// TIA Portal project "Project4" (V17)

(* hardware
DEVICE "S7-1200 station_1"  S7-1200 Station
   slot 0: "Rack_0"  S7-1200 Rack  Rack  V1.0
   slot 1: "PLC_1"  CPU 1214C AC/DC/Rly  6ES7 214-1BG40-0XB0  V4.2
*)

// ===== PLC "PLC_1"  CPU 1214C AC/DC/Rly =====

VAR_GLOBAL   // PLC tag table "Default tag table"
   "PB0" AT %I0.0 : Bool;
   "PB1" AT %I0.1 : Bool;
   "PB2" AT %I0.2 : Bool;
   "PB3" AT %I0.3 : Bool;
   "PB4" AT %I0.4 : Bool;
   "PB5" AT %I0.5 : Bool;
   "PL1" AT %Q0.0 : Bool;
   "PL2" AT %Q0.1 : Bool;
   "PL3" AT %Q0.2 : Bool;
   "PL4" AT %Q0.3 : Bool;
   "X1" AT %M0.0 : Bool;
   "X2" AT %M0.1 : Bool;
   "X3" AT %M0.2 : Bool;
   "X4" AT %M0.3 : Bool;
   "X5" AT %M0.4 : Bool;
   "Tag_1" AT %M10.0 : Bool;
END_VAR

ORGANIZATION_BLOCK "Main"   // OB1, LAD, ProgramCycle
TITLE = "Main Program Sweep (Cycle)"
{ S7_Optimized_Access := 'TRUE' }
VERSION : 0.1
   VAR_INPUT
      Initial_Call : Bool;   // Initial call of this OB
      Remanence : Bool;   // =True, if remanent data are available
   END_VAR
   VAR_TEMP   // added for the SCL form of the ladder/FBD networks
      _w1 : Bool;
   END_VAR
BEGIN

REGION Network 1
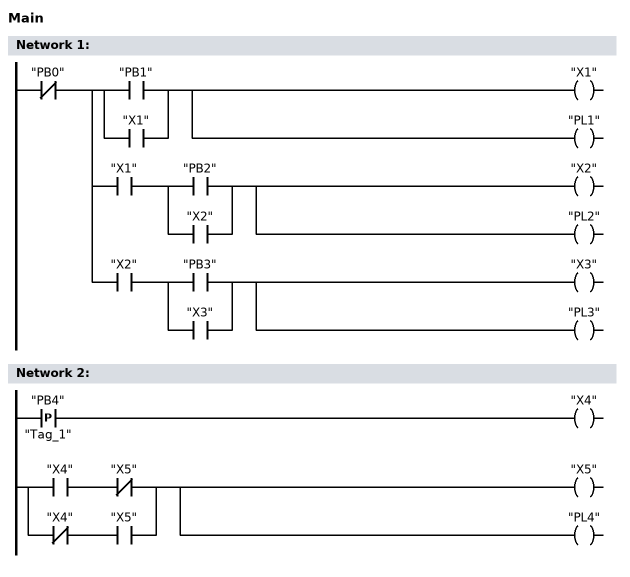
   RUNG wire#powerrail
      I_Contact( "PB0" )
      wire#w1
      Contact( "PB1" )
      wire#w2
      Coil( "X1" )
   END_RUNG
   RUNG wire#w1
      Contact( "X1" )
   END_RUNG wire#w2
   RUNG wire#w2
      Coil( "PL1" )
   END_RUNG
   RUNG wire#w1
      Contact( "X1" )
      wire#w3
      Contact( "PB2" )
      wire#w4
      Coil( "X2" )
   END_RUNG
   RUNG wire#w3
      Contact( "X2" )
   END_RUNG wire#w4
   RUNG wire#w4
      Coil( "PL2" )
   END_RUNG
   RUNG wire#w1
      Contact( "X2" )
      wire#w5
      Contact( "PB3" )
      wire#w6
      Coil( "X3" )
   END_RUNG
   RUNG wire#w5
      Contact( "X3" )
   END_RUNG wire#w6
   RUNG wire#w6
      Coil( "PL3" )
   END_RUNG
   // the same network as SCL:
   "X1" := NOT "PB0" AND ("PB1" OR "X1");
   "PL1" := "X1";
   "X2" := NOT "PB0" AND "X1" AND ("PB2" OR "X2");
   "PL2" := "X2";
   "X3" := NOT "PB0" AND "X2" AND ("PB3" OR "X3");
   "PL3" := "X3";
END_REGION

REGION Network 2
   RUNG wire#powerrail
      P_Contact(operand := "PB4", bit := "Tag_1")
      Coil( "X4" )
   END_RUNG
   RUNG wire#powerrail
      Contact( "X4" )
      I_Contact( "X5" )
      wire#w1
      Coil( "X5" )
   END_RUNG
   RUNG wire#powerrail
      I_Contact( "X4" )
      Contact( "X5" )
   END_RUNG wire#w1
   RUNG wire#w1
      Coil( "PL4" )
   END_RUNG
   // the same network as SCL:
   #_w1 := "PB4" AND NOT "Tag_1";   // rising edge of "PB4"
   "Tag_1" := "PB4";
   "X4" := #_w1;
   "X5" := ("X4" AND NOT "X5") OR (NOT "X4" AND "X5");
   "PL4" := "X5";
END_REGION
END_ORGANIZATION_BLOCK